# EPICS substitutions: apps/mmfeuApp/Db/mmfeuslotAHDC.substitutions
#
file "db/mmfeuslot.db" {
        pattern { P, C, S, PORT}
                {"B_DET_AHDC_FEU", "1",  "1", "L1"}
                {"B_DET_AHDC_FEU", "1",  "2", "L1"}
                {"B_DET_AHDC_FEU", "2",  "1", "L1"}
                {"B_DET_AHDC_FEU", "2",  "2", "L1"}
                {"B_DET_AHDC_FEU", "3",  "1", "L1"}
                {"B_DET_AHDC_FEU", "3",  "2", "L1"}
}
